// TwinCAT 3 PLC project smallproject
// ProgramVersion: 3.1.4024.0
// libraries:
//   Tc2_Standard, * (Beckhoff Automation GmbH)
//   Tc2_System, * (Beckhoff Automation GmbH)
//   Tc3_Module, * (Beckhoff Automation GmbH)
// project tree:
//   DUTs/ DUTSample.TcDUT
//   GVLs/ GLOBAL.TcGVL
//   / PlcTask.TcTTO
//   POUs/ MAIN.TcPOU
// real-time tasks:
//   TASK 2ms: cycle T#2ms, priority 3, ADS port 350
//   TASK 10ms: cycle T#10ms, priority 4, ADS port 351
//   TASK 200ms: cycle T#200000us, priority 6, ADS port 352
//   TASK FileWriterTask: cycle T#200000us, priority 1, ADS port 353
//   TASK PlcTask: cycle T#10ms, priority 20, ADS port 354
// I/O:
//   DEVICE Device 1 (EtherCAT) (disabled), AmsNetId 0.0.0.0.2.1
//     TermEtherCAT (EK1200) [EK1200-5000 EtherCAT Power supply (2A E-Bus)]
//       TermPower1 (EL9222-5500) [EL9222-5500 Overcurrent protection 24V DC, 2Ch., max. 10A (sum), adjustable]
//       TermOutput (EL2008) [EL2008 8Ch. Dig. Output 24V, 0.5A]
//       TermSensorGnrl (EL6224) [EL6224 (IO Link Master)]
//       TermPower2 (EL9222-5500) [EL9222-5500 Overcurrent protection 24V DC, 2Ch., max. 10A (sum), adjustable]
//       TermSensorFront (EL6224) [EL6224 (IO Link Master)]
//       TermSensorBack (EL6224) [EL6224 (IO Link Master)]
//       TermSensorEndstop (EL6224) [EL6224 (IO Link Master)]
//       Pr [EL6224 (IO Link Master)]
//       TermSafety (EL2911) [EL2911, Potential supply terminal (10 A) with 4 Ch. Safety Inputs, TwinSAFE]
//         modules: Module 2 (FSOUT), Module 3 (DEVICEIO), Module 4 (FSLOGIC)
//     Term 31 (EL3062) [EL3062 2Ch. Ana. Input 0-10V]
//     Term 32 (EL9505) [EL9505 Power supply terminal 5V]
//     Term 18 (EL9011) [EL9011 End Terminal]
//   DEVICE CanopenMaster (disabled), AmsNetId 0.0.0.0.6.1
//     DriveLnMn_15
//     Lift_18_Brake
//     DriveMain_17
//     DriveLane_16
//     Bms_32

CONFIGURATION smallproject
    RESOURCE PLC ON TwinCAT3
        TASK PlcTask(INTERVAL := T#10ms, PRIORITY := 20);
        PROGRAM MAIN WITH PlcTask : MAIN;
    END_RESOURCE
END_CONFIGURATION

// ---- DUTs/DUTSample.TcDUT
TYPE DUTSample :
STRUCT
    Counter : INT;
    Ready   : BOOL;
	gIntArray : ARRAY[0..50] OF INT;  
END_STRUCT
END_TYPE

// ---- GVLs/GLOBAL.TcGVL
{attribute 'qualified_only'}
VAR_GLOBAL
	gMyInt: INT := 0;
    gMyBool : BOOL;
	gMyDINT : DINT;
	
	gMyIntCounter : INT := 0;
	gMyBoolToogle : BOOL := FALSE;
	
	gIntCounterActive : BOOL := TRUE;
	gBoolToggleActive : BOOL := TRUE;
	
	// Period used by the timed logic (modifiable via ADS)
    gCyclePeriod      : TIME := T#2S;
	
	// -----------------------
	
	gTimedIntCounter : INT := 0;
	gTimedBoolToogle : BOOL := FALSE;
	
	gTimedCounterActive : BOOL := TRUE;
	gTimedToggleActive : BOOL := TRUE;
	
	 gIntArray : ARRAY[0..100] OF INT;  

	gMyDUT : DUTSample;

END_VAR

// ---- POUs/MAIN.TcPOU
PROGRAM MAIN
VAR
	fbTimer : TON;
    bTick   : BOOL;

END_VAR


// ------------------------------------------------------------
// A) Cycle-based behavior (each PLC scan)
// ------------------------------------------------------------

IF GLOBAL.gIntCounterActive THEN
    GLOBAL.gMyIntCounter := GLOBAL.gMyIntCounter + 1;
END_IF

IF GLOBAL.gBoolToggleActive THEN
    GLOBAL.gMyBoolToogle := NOT GLOBAL.gMyBoolToogle;
END_IF

// ------------------------------------------------------------
// B) Time-based behavior (every gCyclePeriod)
// This triggers a "tick" each time the TON elapses.
// ------------------------------------------------------------
fbTimer(IN := TRUE, PT := GLOBAL.gCyclePeriod);

// bTick is TRUE only when timer is done
bTick := fbTimer.Q;

IF bTick THEN
    // Do the same actions, but only on the tick
    IF GLOBAL.gTimedCounterActive THEN
        GLOBAL.gTimedIntCounter := GLOBAL.gTimedIntCounter + 1;
    END_IF

    IF GLOBAL.gTimedToggleActive THEN
        GLOBAL.gTimedBoolToogle := NOT GLOBAL.gTimedBoolToogle;
    END_IF

    // Retrigger timer (create a periodic pulse)
    fbTimer(IN := FALSE);
END_IF

END_PROGRAM
